(* Logix 5000 project; controller VET 1756-L62 rev 19.52; software revision 19.01; part 19 of 27 *)
(* tags used below, declared in another part *)
   _reset_local : ALIAS FOR _reset_locales.1;
   dsf_l : set_variables;   // Var. Dosificación Líquidos
   dsf_s : set_variables;   // Var. Dosificación Sólidos
   estado : DINT[10];
   _Eqp : Equipo[800];
   _Parametros_D : DINT[30];
   _Parametros_F : REAL[30];
   Batch : batch[10];
   Batch_buff : batch;
   comandos : DINT[10];
   corriente : REAL[40];
   db_input_cola_batch_res : DINT;
   dosificador : dosif_struct[20];
   peso_tolva : REAL[80];
   TabDosif : tabDosif;
   vdf : VDFS[20];
(* Gestion_Dosificacion, continued *)

ROUTINE Gestion_Liquidos_Listos   (* ladder *)
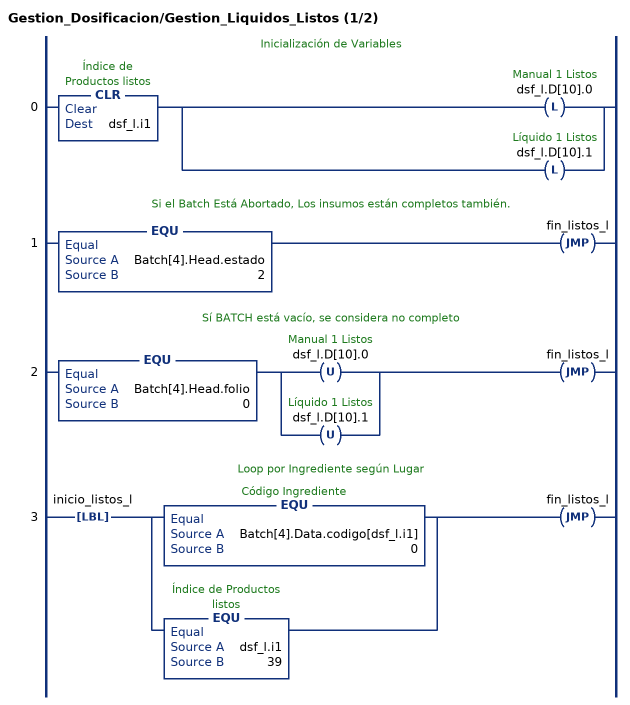
   // Inicialización de Variables
   0: CLR(dsf_l.i1)[OTL(dsf_l.D[10].0) ,OTL(dsf_l.D[10].1) ];
   // Si el Batch Está Abortado, Los insumos están completos también.
   1: EQU(Batch[4].Head.estado,2)JMP(fin_listos_l);
   // Sí BATCH está vacío, se considera no completo
   2: EQU(Batch[4].Head.folio,0)[OTU(dsf_l.D[10].0) ,OTU(dsf_l.D[10].1) ]JMP(fin_listos_l);
   // Loop por Ingrediente según Lugar
   3: LBL(inicio_listos_l)[EQU(Batch[4].Data.codigo[dsf_l.i1],0) ,EQU(dsf_l.i1,39) ]JMP(fin_listos_l);
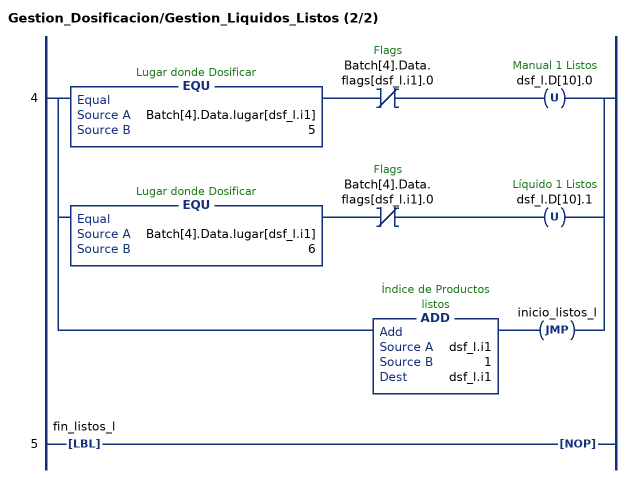
   4: [EQU(Batch[4].Data.lugar[dsf_l.i1],5) XIO(Batch[4].Data.flags[dsf_l.i1].0) OTU(dsf_l.D[10].0) ,EQU(Batch[4].Data.lugar[dsf_l.i1],6) XIO(Batch[4].Data.flags[dsf_l.i1].0) OTU(dsf_l.D[10].1) ,ADD(dsf_l.i1,1,dsf_l.i1) JMP(inicio_listos_l) ];
   5: LBL(fin_listos_l)NOP();
END_ROUTINE

ROUTINE Gestion_Loop_Ingredientes_Liquidos   (* ladder *)
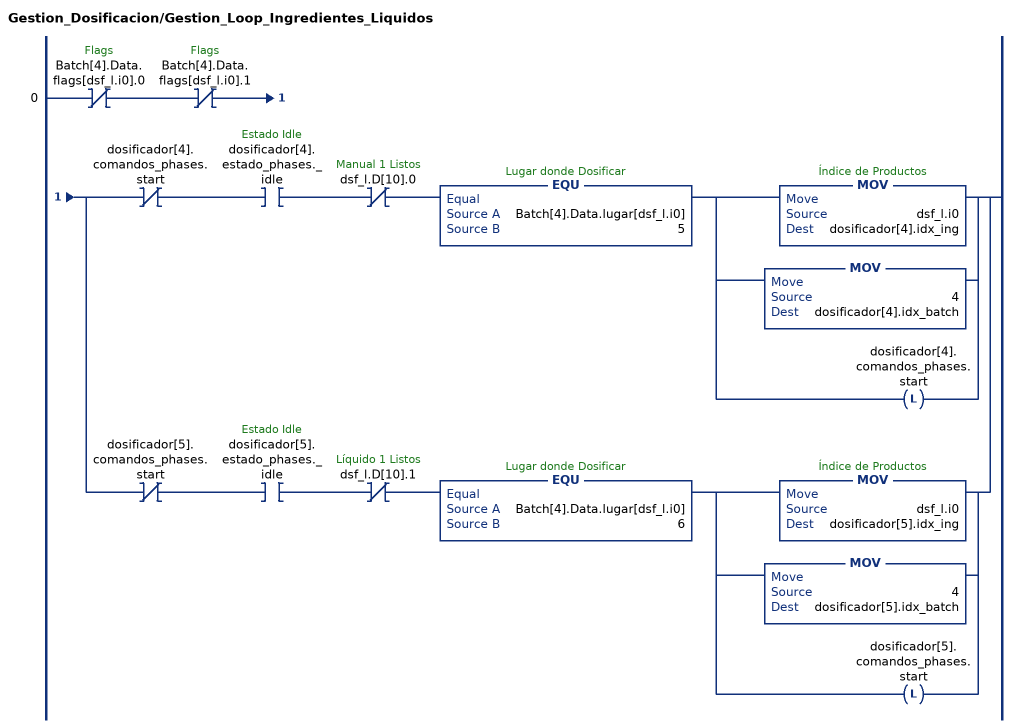
   0: XIO(Batch[4].Data.flags[dsf_l.i0].0)XIO(Batch[4].Data.flags[dsf_l.i0].1)[XIO(dosificador[4].comandos_phases.start) XIC(dosificador[4].estado_phases._idle) XIO(dsf_l.D[10].0) EQU(Batch[4].Data.lugar[dsf_l.i0],5) [MOV(dsf_l.i0,dosificador[4].idx_ing) ,MOV(4,dosificador[4].idx_batch) ,OTL(dosificador[4].comandos_phases.start) ] ,XIO(dosificador[5].comandos_phases.start) XIC(dosificador[5].estado_phases._idle) XIO(dsf_l.D[10].1) EQU(Batch[4].Data.lugar[dsf_l.i0],6) [MOV(dsf_l.i0,dosificador[5].idx_ing) ,MOV(4,dosificador[5].idx_batch) ,OTL(dosificador[5].comandos_phases.start) ] ];
END_ROUTINE

ROUTINE Gestion_Loop_Ingredientes_Solidos   (* ladder *)
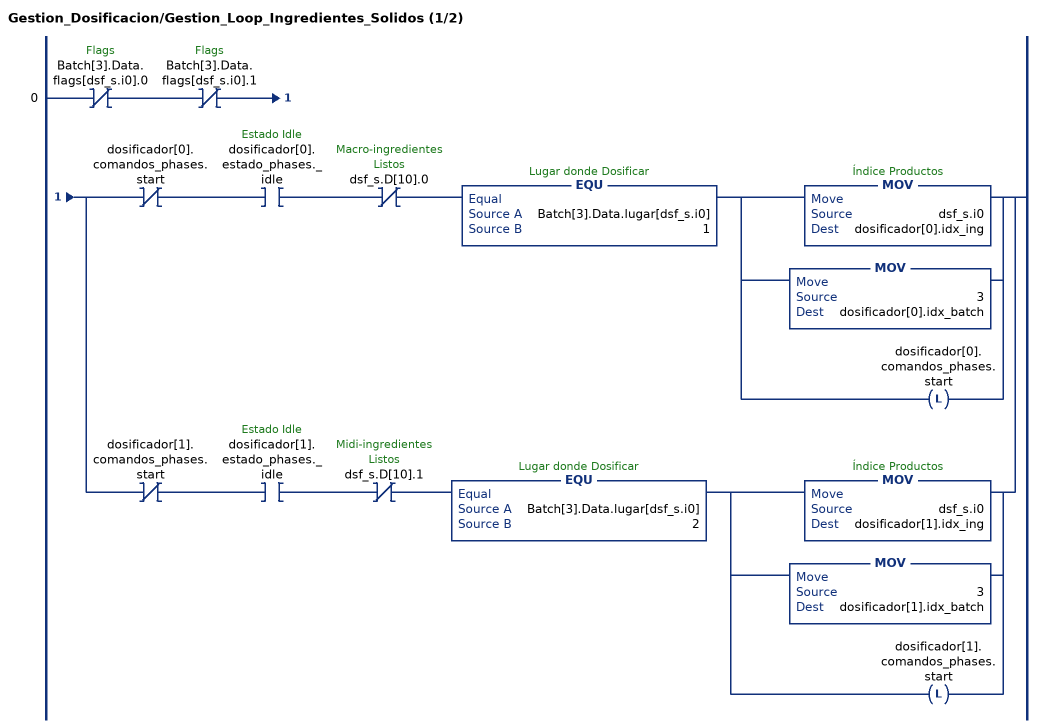
   0: XIO(Batch[3].Data.flags[dsf_s.i0].0)XIO(Batch[3].Data.flags[dsf_s.i0].1)[XIO(dosificador[0].comandos_phases.start) XIC(dosificador[0].estado_phases._idle) XIO(dsf_s.D[10].0) EQU(Batch[3].Data.lugar[dsf_s.i0],1) [MOV(dsf_s.i0,dosificador[0].idx_ing) ,MOV(3,dosificador[0].idx_batch) ,OTL(dosificador[0].comandos_phases.start) ] ,XIO(dosificador[1].comandos_phases.start) XIC(dosificador[1].estado_phases._idle) XIO(dsf_s.D[10].1) EQU(Batch[3].Data.lugar[dsf_s.i0],2) [MOV(dsf_s.i0,dosificador[1].idx_ing) ,MOV(3,dosificador[1].idx_batch) ,OTL(dosificador[1].comandos_phases.start) ] ];
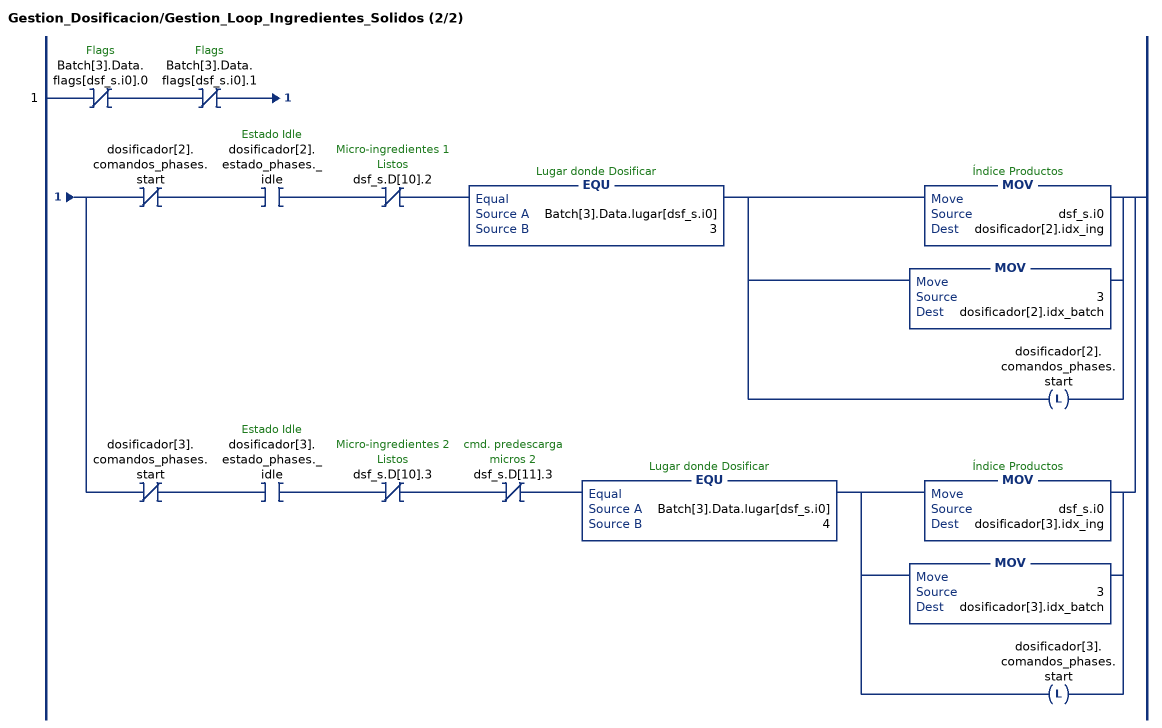
   1: XIO(Batch[3].Data.flags[dsf_s.i0].0)XIO(Batch[3].Data.flags[dsf_s.i0].1)[XIO(dosificador[2].comandos_phases.start) XIC(dosificador[2].estado_phases._idle) XIO(dsf_s.D[10].2) EQU(Batch[3].Data.lugar[dsf_s.i0],3) [MOV(dsf_s.i0,dosificador[2].idx_ing) ,MOV(3,dosificador[2].idx_batch) ,OTL(dosificador[2].comandos_phases.start) ] ,XIO(dosificador[3].comandos_phases.start) XIC(dosificador[3].estado_phases._idle) XIO(dsf_s.D[10].3) XIO(dsf_s.D[11].3) EQU(Batch[3].Data.lugar[dsf_s.i0],4) [MOV(dsf_s.i0,dosificador[3].idx_ing) ,MOV(3,dosificador[3].idx_batch) ,OTL(dosificador[3].comandos_phases.start) ] ];
END_ROUTINE

ROUTINE Gestion_Solidos   (* ladder *)
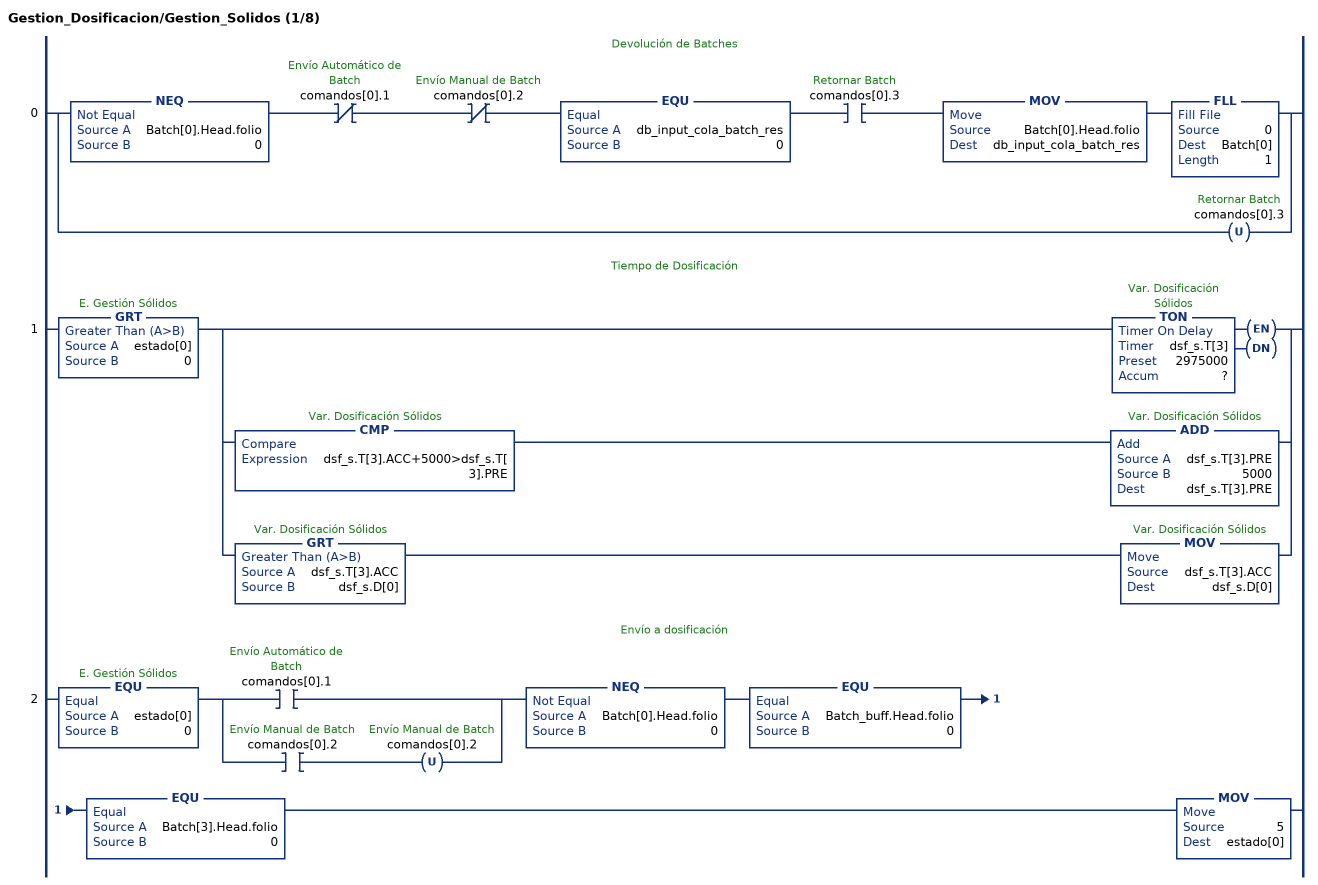
   // Devolución de Batches
   0: [NEQ(Batch[0].Head.folio,0) XIO(comandos[0].1) XIO(comandos[0].2) EQU(db_input_cola_batch_res,0) XIC(comandos[0].3) MOV(Batch[0].Head.folio,db_input_cola_batch_res) FLL(0,Batch[0],1) ,OTU(comandos[0].3) ];
   // Tiempo de Dosificación
   1: GRT(estado[0],0)[TON(dsf_s.T[3],?,?) ,CMP(dsf_s.T[3].ACC+5000>dsf_s.T[3].PRE) ADD(dsf_s.T[3].PRE,5000,dsf_s.T[3].PRE) ,GRT(dsf_s.T[3].ACC,dsf_s.D[0]) MOV(dsf_s.T[3].ACC,dsf_s.D[0]) ];
   // Envío a dosificación
   2: EQU(estado[0],0)[XIC(comandos[0].1) ,XIC(comandos[0].2) OTU(comandos[0].2) ]NEQ(Batch[0].Head.folio,0)EQU(Batch_buff.Head.folio,0)EQU(Batch[3].Head.folio,0)MOV(5,estado[0]);
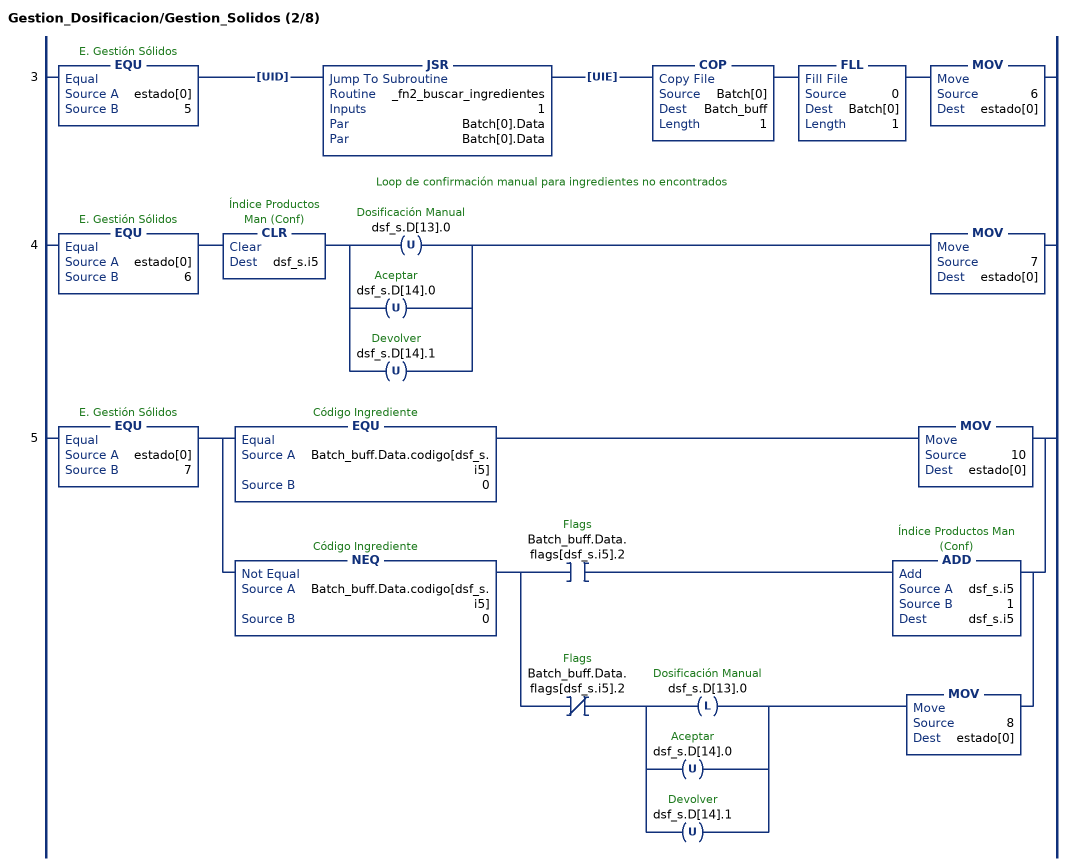
   3: EQU(estado[0],5)UID()JSR(_fn2_buscar_ingredientes,1,Batch[0].Data,Batch[0].Data)UIE()COP(Batch[0],Batch_buff,1)FLL(0,Batch[0],1)MOV(6,estado[0]);
   // Loop de confirmación manual para ingredientes no encontrados
   4: EQU(estado[0],6)CLR(dsf_s.i5)[OTU(dsf_s.D[13].0) ,OTU(dsf_s.D[14].0) ,OTU(dsf_s.D[14].1) ]MOV(7,estado[0]);
   5: EQU(estado[0],7)[EQU(Batch_buff.Data.codigo[dsf_s.i5],0) MOV(10,estado[0]) ,NEQ(Batch_buff.Data.codigo[dsf_s.i5],0) [XIC(Batch_buff.Data.flags[dsf_s.i5].2) ADD(dsf_s.i5,1,dsf_s.i5) ,XIO(Batch_buff.Data.flags[dsf_s.i5].2) [OTL(dsf_s.D[13].0) ,OTU(dsf_s.D[14].0) ,OTU(dsf_s.D[14].1) ] MOV(8,estado[0]) ] ];
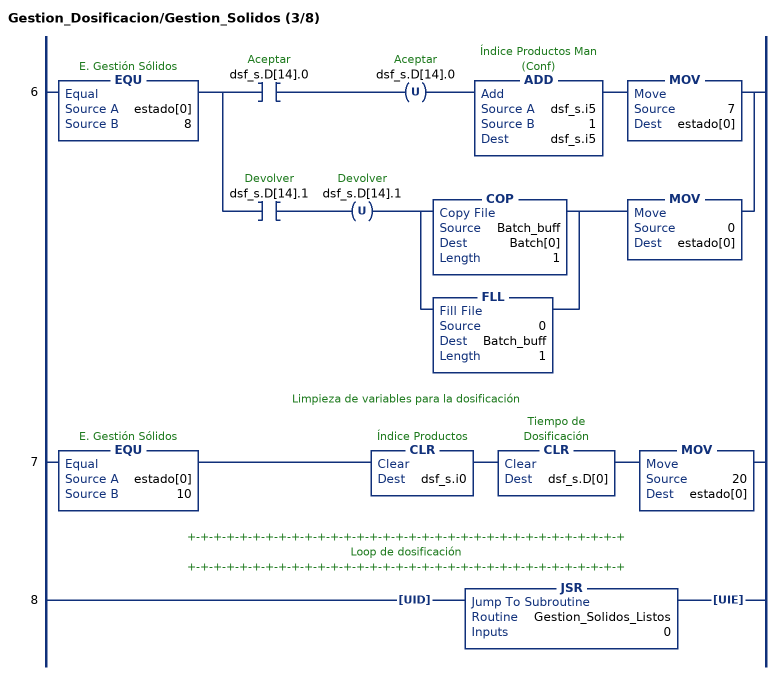
   6: EQU(estado[0],8)[XIC(dsf_s.D[14].0) OTU(dsf_s.D[14].0) ADD(dsf_s.i5,1,dsf_s.i5) MOV(7,estado[0]) ,XIC(dsf_s.D[14].1) OTU(dsf_s.D[14].1) [COP(Batch_buff,Batch[0],1) ,FLL(0,Batch_buff,1) ] MOV(0,estado[0]) ];
   // Limpieza de variables para la dosificación
   7: EQU(estado[0],10)CLR(dsf_s.i0)CLR(dsf_s.D[0])MOV(20,estado[0]);
   // +-+-+-+-+-+-+-+-+-+-+-+-+-+-+-+-+-+-+-+-+-+-+-+-+-+-+-+-+-+-+-+-+-+
   // Loop de dosificación
   // +-+-+-+-+-+-+-+-+-+-+-+-+-+-+-+-+-+-+-+-+-+-+-+-+-+-+-+-+-+-+-+-+-+
   8: UID()JSR(Gestion_Solidos_Listos,0)UIE();
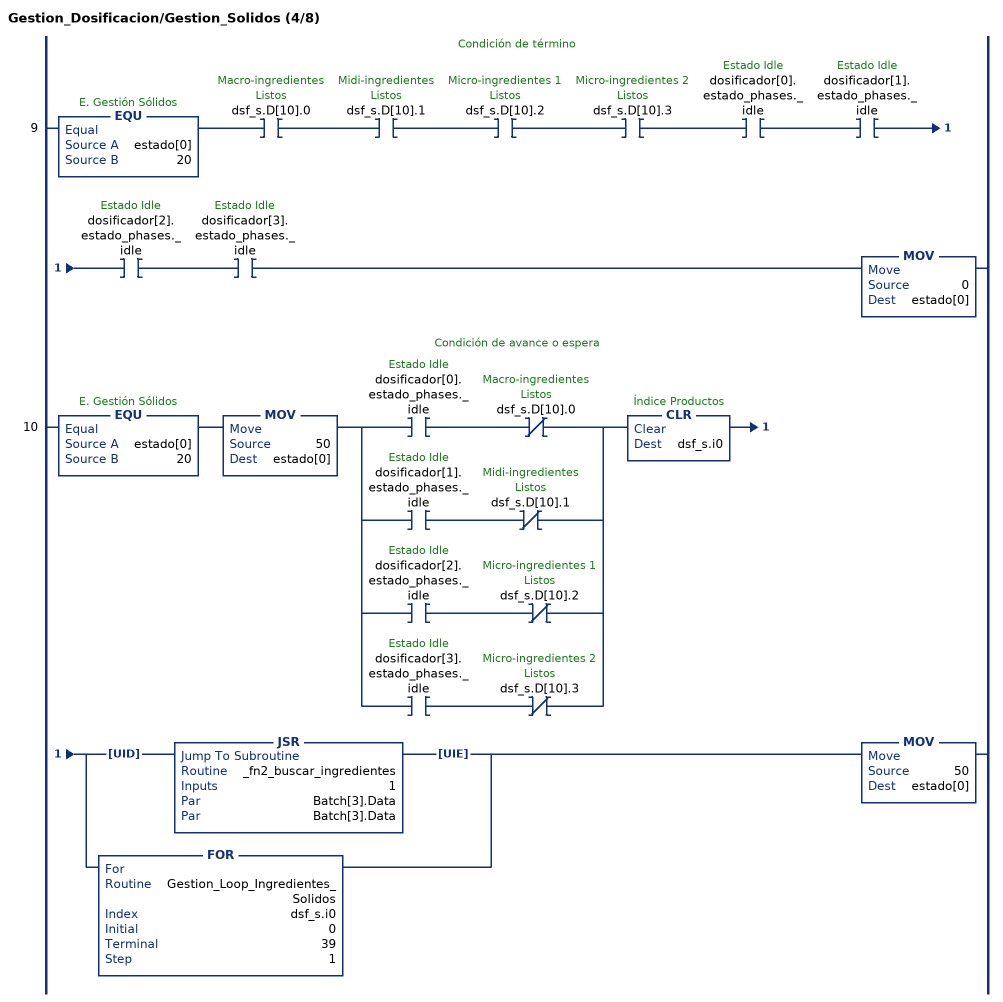
   // Condición de término
   9: EQU(estado[0],20)XIC(dsf_s.D[10].0)XIC(dsf_s.D[10].1)XIC(dsf_s.D[10].2)XIC(dsf_s.D[10].3)XIC(dosificador[0].estado_phases._idle)XIC(dosificador[1].estado_phases._idle)XIC(dosificador[2].estado_phases._idle)XIC(dosificador[3].estado_phases._idle)MOV(0,estado[0]);
   // Condición de avance o espera
   10: EQU(estado[0],20)MOV(50,estado[0])[XIC(dosificador[0].estado_phases._idle) XIO(dsf_s.D[10].0) ,XIC(dosificador[1].estado_phases._idle) XIO(dsf_s.D[10].1) ,XIC(dosificador[2].estado_phases._idle) XIO(dsf_s.D[10].2) ,XIC(dosificador[3].estado_phases._idle) XIO(dsf_s.D[10].3) ]CLR(dsf_s.i0)[UID() JSR(_fn2_buscar_ingredientes,1,Batch[3].Data,Batch[3].Data) UIE() ,FOR(Gestion_Loop_Ingredientes_Solidos,dsf_s.i0,0,39,1) ]MOV(50,estado[0]);
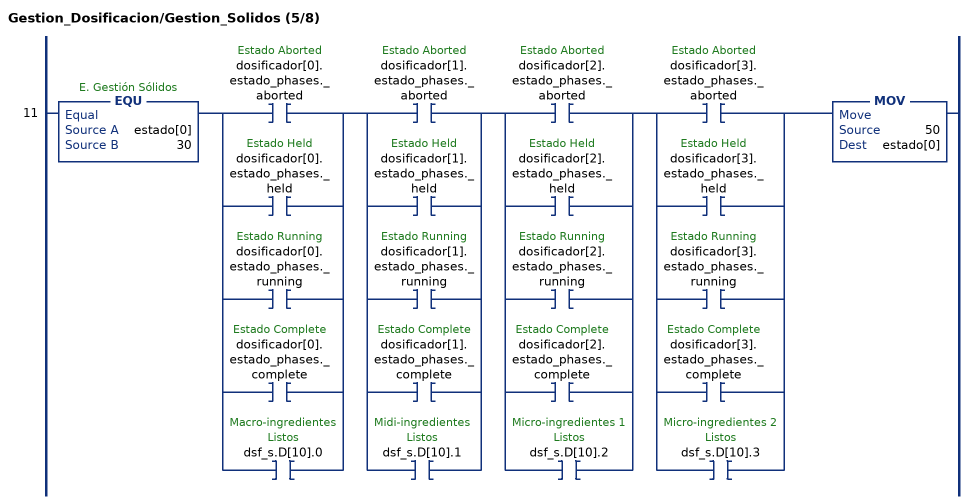
   11: EQU(estado[0],30)[XIC(dosificador[0].estado_phases._aborted) ,XIC(dosificador[0].estado_phases._held) ,XIC(dosificador[0].estado_phases._running) ,XIC(dosificador[0].estado_phases._complete) ,XIC(dsf_s.D[10].0) ][XIC(dosificador[1].estado_phases._aborted) ,XIC(dosificador[1].estado_phases._held) ,XIC(dosificador[1].estado_phases._running) ,XIC(dosificador[1].estado_phases._complete) ,XIC(dsf_s.D[10].1) ][XIC(dosificador[2].estado_phases._aborted) ,XIC(dosificador[2].estado_phases._held) ,XIC(dosificador[2].estado_phases._running) ,XIC(dosificador[2].estado_phases._complete) ,XIC(dsf_s.D[10].2) ][XIC(dosificador[3].estado_phases._aborted) ,XIC(dosificador[3].estado_phases._held) ,XIC(dosificador[3].estado_phases._running) ,XIC(dosificador[3].estado_phases._complete) ,XIC(dsf_s.D[10].3) ]MOV(50,estado[0]);
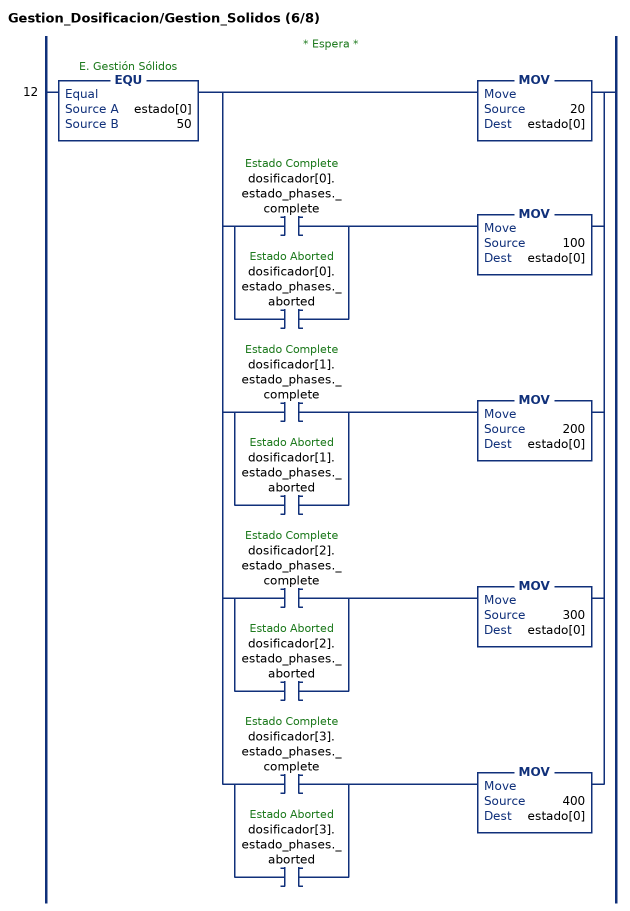
   // * Espera *
   12: EQU(estado[0],50)[MOV(20,estado[0]) ,[XIC(dosificador[0].estado_phases._complete) ,XIC(dosificador[0].estado_phases._aborted) ] MOV(100,estado[0]) ,[XIC(dosificador[1].estado_phases._complete) ,XIC(dosificador[1].estado_phases._aborted) ] MOV(200,estado[0]) ,[XIC(dosificador[2].estado_phases._complete) ,XIC(dosificador[2].estado_phases._aborted) ] MOV(300,estado[0]) ,[XIC(dosificador[3].estado_phases._complete) ,XIC(dosificador[3].estado_phases._aborted) ] MOV(400,estado[0]) ];
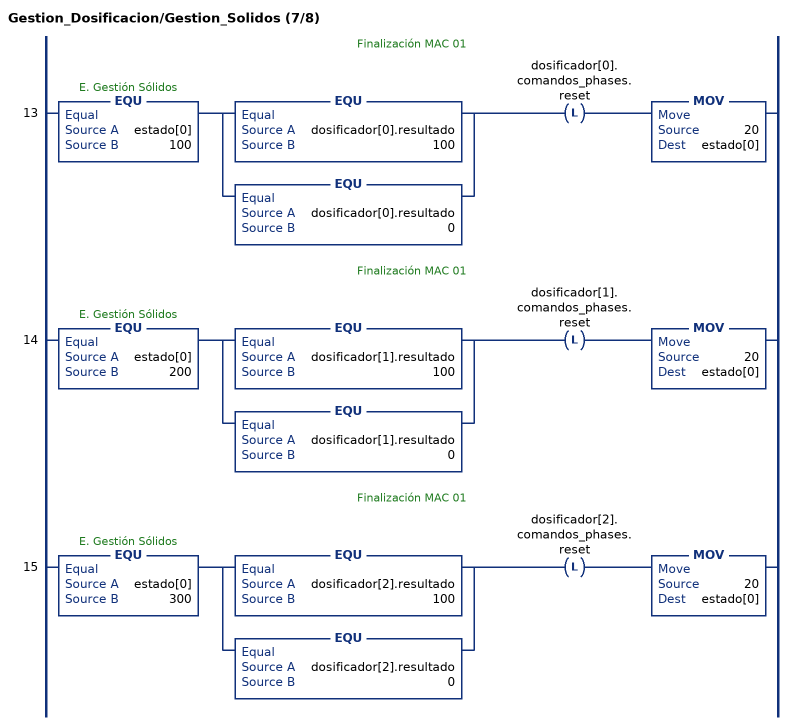
   // Finalización MAC 01
   13: EQU(estado[0],100)[EQU(dosificador[0].resultado,100) ,EQU(dosificador[0].resultado,0) ]OTL(dosificador[0].comandos_phases.reset)MOV(20,estado[0]);
   // Finalización MAC 01
   14: EQU(estado[0],200)[EQU(dosificador[1].resultado,100) ,EQU(dosificador[1].resultado,0) ]OTL(dosificador[1].comandos_phases.reset)MOV(20,estado[0]);
   // Finalización MAC 01
   15: EQU(estado[0],300)[EQU(dosificador[2].resultado,100) ,EQU(dosificador[2].resultado,0) ]OTL(dosificador[2].comandos_phases.reset)MOV(20,estado[0]);
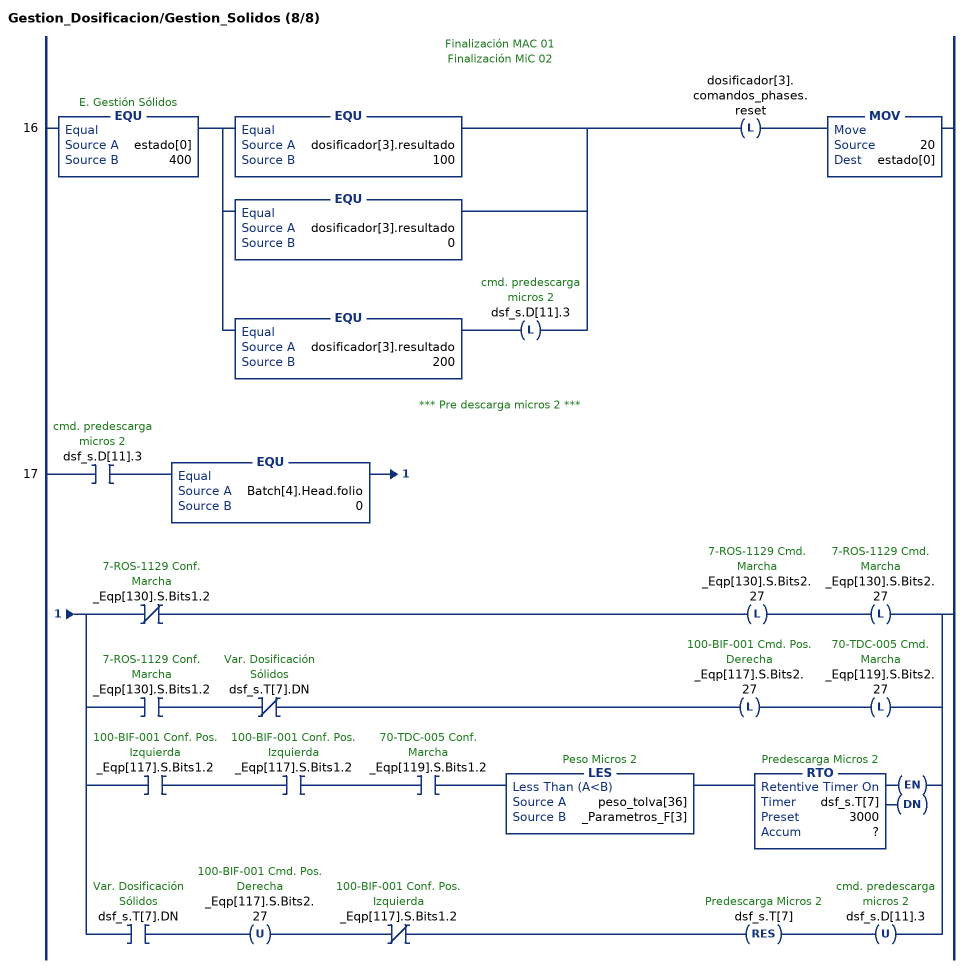
   // Finalización MAC 01
   // Finalización MiC 02
   16: EQU(estado[0],400)[EQU(dosificador[3].resultado,100) ,EQU(dosificador[3].resultado,0) ,EQU(dosificador[3].resultado,200) OTL(dsf_s.D[11].3) ]OTL(dosificador[3].comandos_phases.reset)MOV(20,estado[0]);
   // *** Pre descarga micros 2 ***
   17: XIC(dsf_s.D[11].3)EQU(Batch[4].Head.folio,0)[XIO(_Eqp[130].S.Bits1.2) OTL(_Eqp[130].S.Bits2.27) OTL(_Eqp[130].S.Bits2.27) ,XIC(_Eqp[130].S.Bits1.2) XIO(dsf_s.T[7].DN) OTL(_Eqp[117].S.Bits2.27) OTL(_Eqp[119].S.Bits2.27) ,XIC(_Eqp[117].S.Bits1.2) XIC(_Eqp[117].S.Bits1.2) XIC(_Eqp[119].S.Bits1.2) LES(peso_tolva[36],_Parametros_F[3]) RTO(dsf_s.T[7],?,?) ,XIC(dsf_s.T[7].DN) OTU(_Eqp[117].S.Bits2.27) XIO(_Eqp[117].S.Bits1.2) RES(dsf_s.T[7]) OTU(dsf_s.D[11].3) ];
END_ROUTINE

ROUTINE Gestion_Solidos_Listos   (* ladder *)
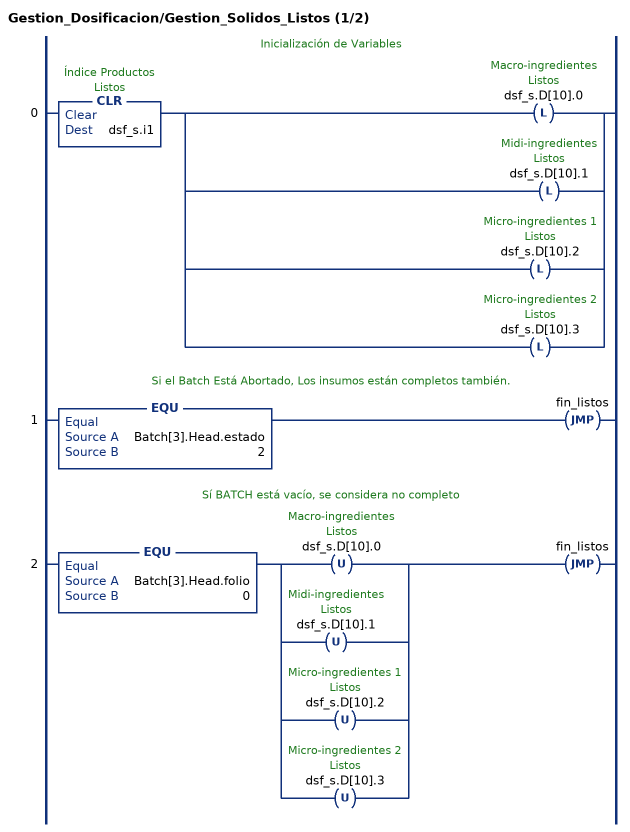
   // Inicialización de Variables
   0: CLR(dsf_s.i1)[OTL(dsf_s.D[10].0) ,OTL(dsf_s.D[10].1) ,OTL(dsf_s.D[10].2) ,OTL(dsf_s.D[10].3) ];
   // Si el Batch Está Abortado, Los insumos están completos también.
   1: EQU(Batch[3].Head.estado,2)JMP(fin_listos);
   // Sí BATCH está vacío, se considera no completo
   2: EQU(Batch[3].Head.folio,0)[OTU(dsf_s.D[10].0) ,OTU(dsf_s.D[10].1) ,OTU(dsf_s.D[10].2) ,OTU(dsf_s.D[10].3) ]JMP(fin_listos);
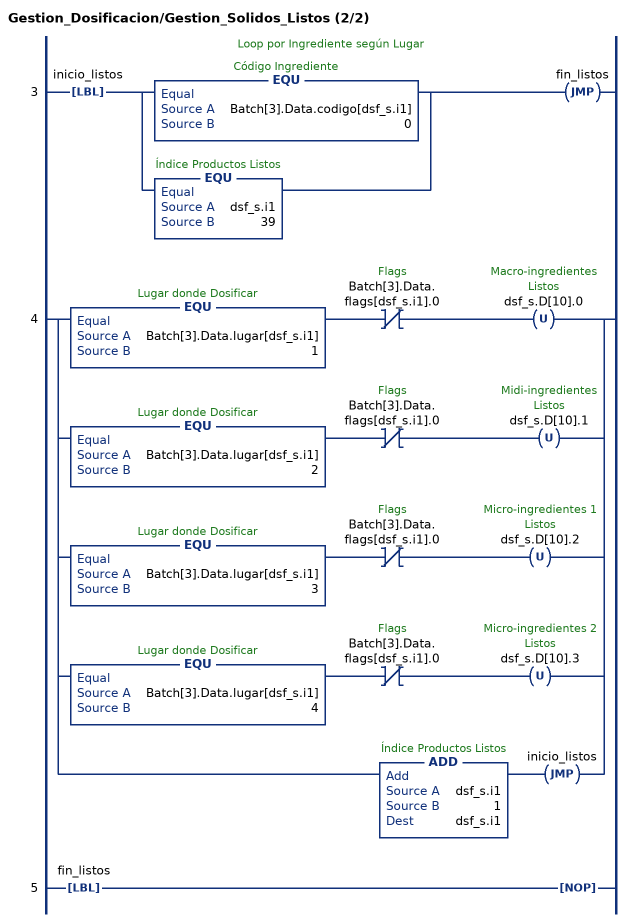
   // Loop por Ingrediente según Lugar
   3: LBL(inicio_listos)[EQU(Batch[3].Data.codigo[dsf_s.i1],0) ,EQU(dsf_s.i1,39) ]JMP(fin_listos);
   4: [EQU(Batch[3].Data.lugar[dsf_s.i1],1) XIO(Batch[3].Data.flags[dsf_s.i1].0) OTU(dsf_s.D[10].0) ,EQU(Batch[3].Data.lugar[dsf_s.i1],2) XIO(Batch[3].Data.flags[dsf_s.i1].0) OTU(dsf_s.D[10].1) ,EQU(Batch[3].Data.lugar[dsf_s.i1],3) XIO(Batch[3].Data.flags[dsf_s.i1].0) OTU(dsf_s.D[10].2) ,EQU(Batch[3].Data.lugar[dsf_s.i1],4) XIO(Batch[3].Data.flags[dsf_s.i1].0) OTU(dsf_s.D[10].3) ,ADD(dsf_s.i1,1,dsf_s.i1) JMP(inicio_listos) ];
   5: LBL(fin_listos)NOP();
END_ROUTINE

ROUTINE Gestion_Transporte_Despacho   (* ladder *)
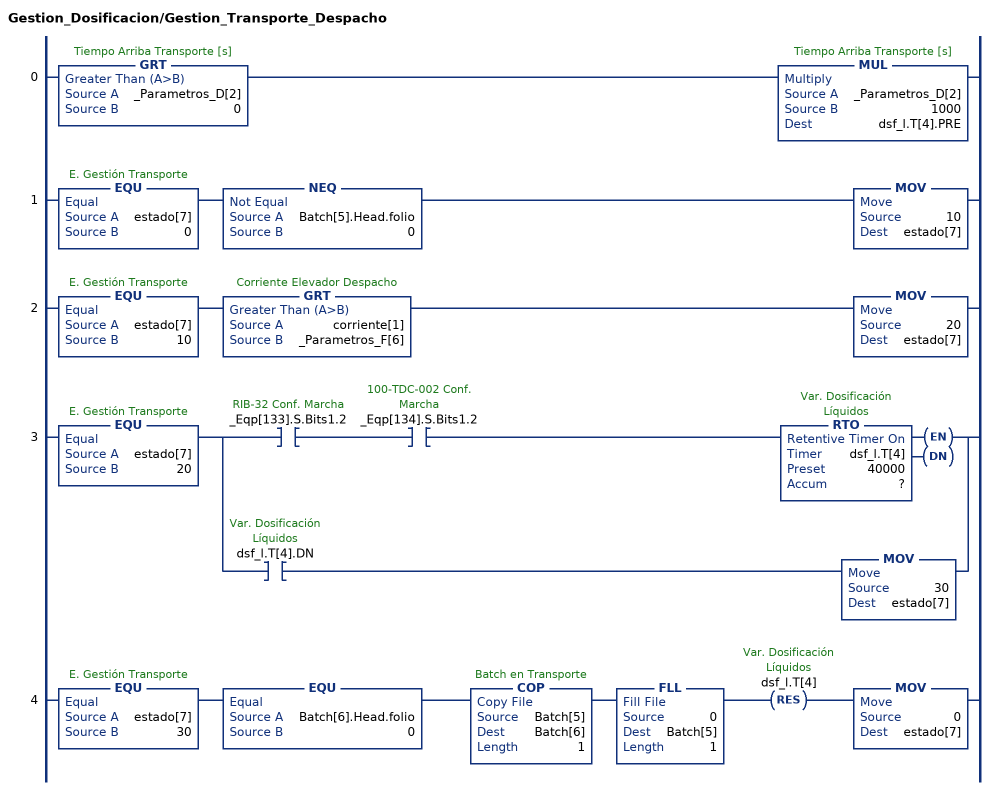
   0: GRT(_Parametros_D[2],0)MUL(_Parametros_D[2],1000,dsf_l.T[4].PRE);
   1: EQU(estado[7],0)NEQ(Batch[5].Head.folio,0)MOV(10,estado[7]);
   2: EQU(estado[7],10)GRT(corriente[1],_Parametros_F[6])MOV(20,estado[7]);
   3: EQU(estado[7],20)[XIC(_Eqp[133].S.Bits1.2) XIC(_Eqp[134].S.Bits1.2) RTO(dsf_l.T[4],?,?) ,XIC(dsf_l.T[4].DN) MOV(30,estado[7]) ];
   4: EQU(estado[7],30)EQU(Batch[6].Head.folio,0)COP(Batch[5],Batch[6],1)FLL(0,Batch[5],1)RES(dsf_l.T[4])MOV(0,estado[7]);
END_ROUTINE

ROUTINE Interfaz_IO_dosificadores   (* ladder *)
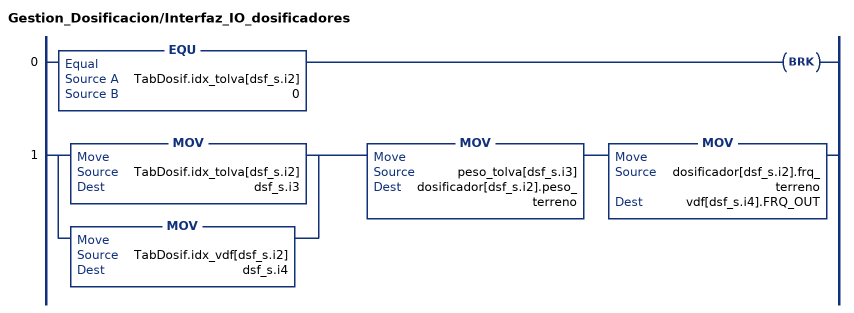
   0: EQU(TabDosif.idx_tolva[dsf_s.i2],0)BRK();
   1: [MOV(TabDosif.idx_tolva[dsf_s.i2],dsf_s.i3) ,MOV(TabDosif.idx_vdf[dsf_s.i2],dsf_s.i4) ]MOV(peso_tolva[dsf_s.i3],dosificador[dsf_s.i2].peso_terreno)MOV(dosificador[dsf_s.i2].frq_terreno,vdf[dsf_s.i4].FRQ_OUT);
END_ROUTINE

ROUTINE Main   (* ladder *)
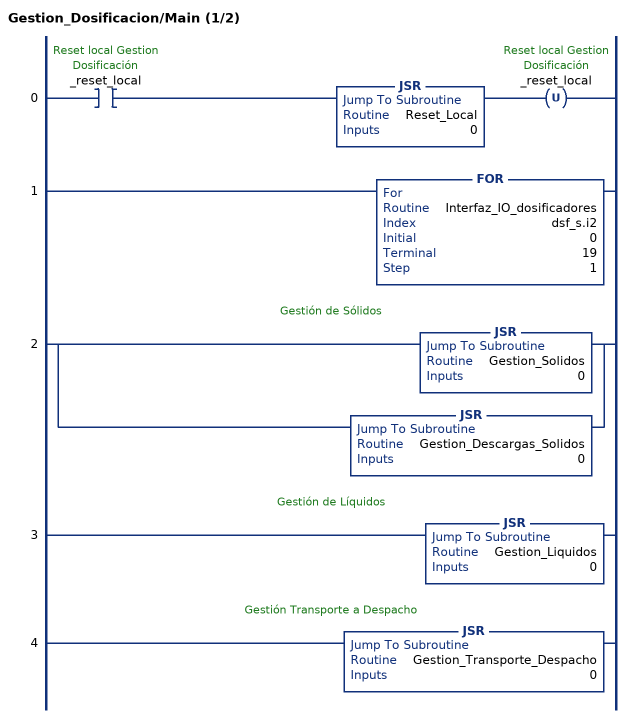
   0: XIC(_reset_local)JSR(Reset_Local,0)OTU(_reset_local);
   1: FOR(Interfaz_IO_dosificadores,dsf_s.i2,0,19,1);
   // Gestión de Sólidos
   2: [JSR(Gestion_Solidos,0) ,JSR(Gestion_Descargas_Solidos,0) ];
   // Gestión de Líquidos
   3: JSR(Gestion_Liquidos,0);
   // Gestión Transporte a Despacho
   4: JSR(Gestion_Transporte_Despacho,0);
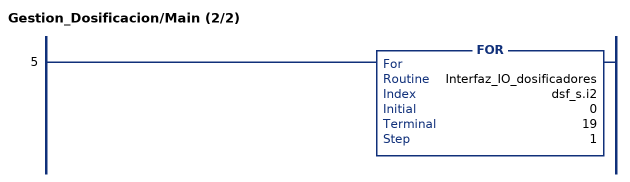
   5: FOR(Interfaz_IO_dosificadores,dsf_s.i2,0,19,1);
END_ROUTINE
